(* PLC project Sin nombre, Desconocido Sin nombre 1 *)
(* stored: creationDateTime 2022-10-17T16:56:25, modificationDateTime 2022-11-07T15:36:23 *)

PROGRAM program0
  VAR
    Out1 AT %QX0.0 : BOOL := 0;  (* Activa o desactiva el pin 1 del motor *)
    Out2 AT %QX0.1 : BOOL := 0;  (* Activa o desactiva el pin 2 del motor *)
    Out3 AT %QX0.2 : BOOL := 0;  (* Activa o desactiva el pin 3 del motor *)
    Out4 AT %QX0.3 : BOOL := 0;  (* Activa o desactiva el pin 4 del motor *)
  END_VAR
  VAR
    demora : TIME := T#15ms;  (* Demora entre cada paso (15 ms = 2 RPM aprox. ) *)
    control : BOOL := 0;  (* Permite cambiar el sentido de giro entre Horario y Antihorario *)
    TP0 : TP;  (* Permite activar el pin 4 del motor *)
    TP1 : TP;  (* Permite activar el pin 3 del motor *)
    TP2 : TP;  (* Permite activar el pin 2 del motor *)
    TP3 : TP;  (* Permite activar el pin 1 del motor *)
    TOF0 : TOF;  (* Permite iniciar nuevamente el ciclo de giro Horario *)
    TP4 : TP;  (* Permite activar el pin 1 del motor *)
    TP5 : TP;  (* Permite activar el pin 2 del motor *)
    TP6 : TP;  (* Permite activar el pin 3 del motor *)
    TP7 : TP;  (* Permite activar el pin 4 del motor *)
    TOF1 : TOF;  (* Permite iniciar nuevamente el ciclo de giro Antihorario *)
  END_VAR

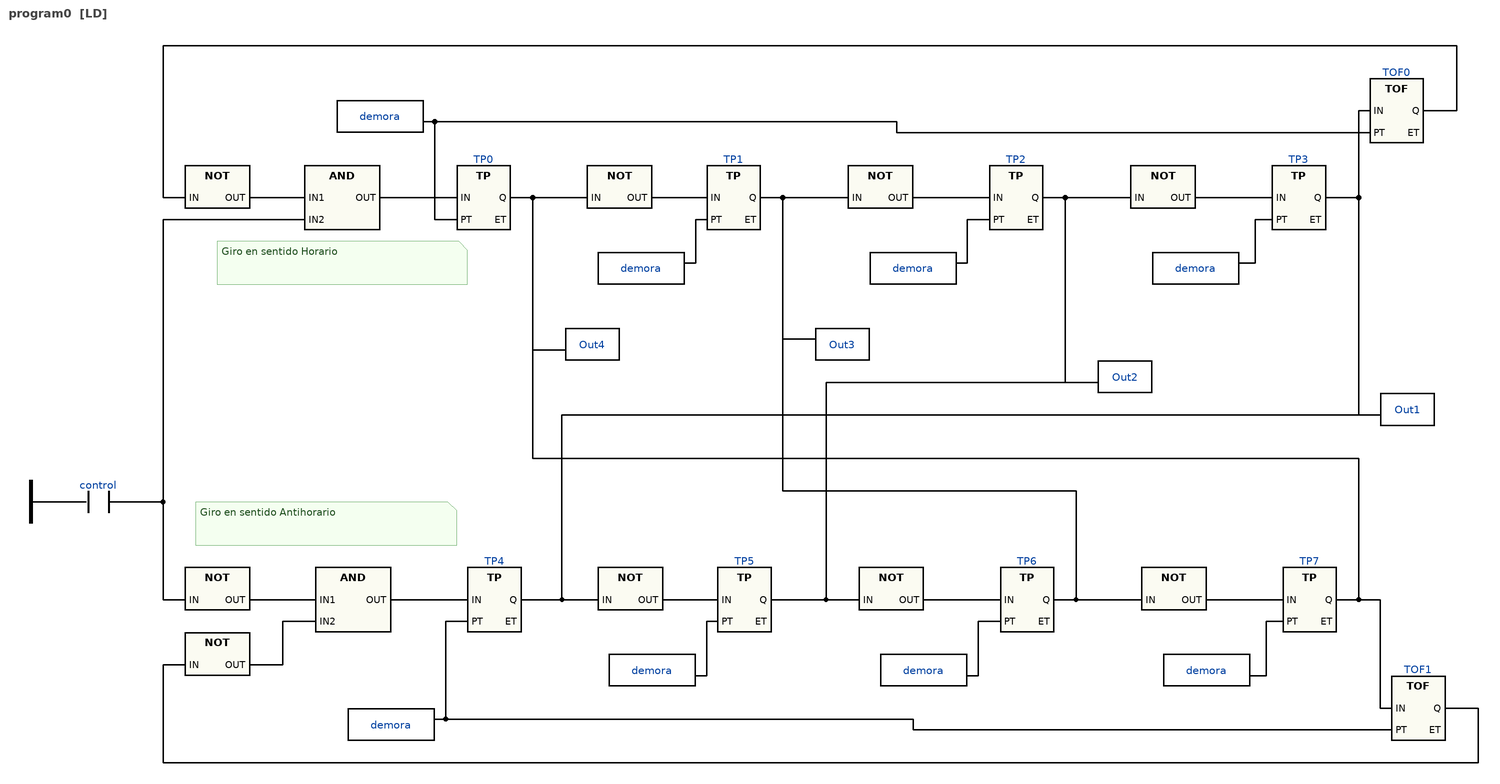
(* LD diagram, written out as Structured Text *)
(* Giro en sentido Horario *)
TP1(IN := NOT TP0.Q, PT := demora);
TP2(IN := NOT TP1.Q, PT := demora);
TP3(IN := NOT TP2.Q, PT := demora);
TOF0(IN := TP3.Q, PT := demora);
TP0(IN := NOT TOF0.Q AND control, PT := demora);
TOF1(IN := TP7.Q, PT := demora);
TP4(IN := NOT control AND NOT TOF1.Q, PT := demora);
TP5(IN := NOT TP4.Q, PT := demora);
TP6(IN := NOT TP5.Q, PT := demora);
TP7(IN := NOT TP6.Q, PT := demora);
Out4 := TP0.Q OR TP7.Q;
Out3 := TP1.Q OR TP6.Q;
Out2 := TP2.Q OR TP5.Q;
Out1 := TP3.Q OR TP4.Q;
(* Giro en sentido Antihorario *)
END_PROGRAM

CONFIGURATION Config0
  RESOURCE Res0 ON PLC
    TASK task0(INTERVAL := T#20ms, PRIORITY := 0);
    PROGRAM instance0 WITH task0 : program0;
  END_RESOURCE
END_CONFIGURATION
